Fanuc KAREL source: CE0150.KL

PROGRAM CE0150
%STACKSIZE=65535
%PRIORITY=65535
%NOLOCKGROUP
ROUTINE RB(P1 : BOOLEAN) : BOOLEAN FROM CE0150
ROUTINE RI(P1 : INTEGER) : INTEGER FROM CE0150
ROUTINE RR(P1 : REAL) : REAL FROM CE0150
ROUTINE RTEST FROM CE0150
ROUTINE RB
BEGIN
RETURN(P1)
-- UNRESOLVED_PC line 6 opcodes [7F] marker_code=16
END RB
ROUTINE RI
BEGIN
-- UNRESOLVED_PC line 9 opcodes [2D 9D 52 7F] marker_code=26
-- UNRESOLVED_PC line 10 opcodes [7F] marker_code=43
END RI
ROUTINE RR
BEGIN
-- UNRESOLVED_PC line 13 opcodes [2D 2E 69 7F] marker_code=53
-- UNRESOLVED_PC line 14 opcodes [7F] marker_code=74
END RR
ROUTINE RTEST
VAR
L1 : STRING[20]
L2 : STRING[20]
L3 : ARRAY[3] OF INTEGER
S1 : INTEGER
U2C_18 : INTEGER -- ASSUMED 2C source type; see uncertainty report
U2C_19 : INTEGER -- ASSUMED 2C source type; see uncertainty report
U2C_20 : INTEGER -- ASSUMED 2C source type; see uncertainty report
S2 : BOOLEAN
U2C_22 : INTEGER -- ASSUMED 2C source type; see uncertainty report
BEGIN
S1=2
U2C_18=3
U2C_19=1075838976
U2C_20=1080033280
S2=TRUE
U2C_22=0
L1='AB'
L2='AC'
L3[1]=2
L3[2]=3
-- UNSAFE_SOURCE_IR line 37: CALL_RESULT RB(S2)
S1=(S1 + 1)
S1=(S1 + 2)
END RTEST
BEGIN
RTEST
END CE0150
